FUNCTION_BLOCK FB_Timeout
VAR_INPUT
	match_time 	: TIME;
	max_time	: TIME;
END_VAR
VAR_OUTPUT
	bstop		: BOOL;
END_VAR

//si le temps de match est dépassé, renvoie un signal d'arrêt 
IF match_time >= max_time THEN 
	bstop := TRUE;
ELSE
	bstop := FALSE;
END_IF

END_FUNCTION_BLOCK

(* stored: Version 1.1.0.1, ProductVersion 3.1.4024.11
   POU FB_Timeout: Id {e880bfd7-d935-47b1-8a9e-1e474bbdb3b8}, SpecialFunc None *)
